{attribute 'strict'}
TYPE E_CSVDataExchangerInsertIntoTableState :
(
	CSV_DATA_EXCHANGER_INSERT_INTO_TABLE_OPEN_FILE 							:= 0,
	CSV_DATA_EXCHANGER_INSERT_INTO_TABLE_WAIT_FOR_OPENING					:= 10,	
	CSV_DATA_EXCHANGER_INSERT_INTO_TABLE_CONV_ONE_RECORD_TO_CSV 			:= 20,	
	CSV_DATA_EXCHANGER_INSERT_INTO_TABLE_WRITE_SINGLE_LINE					:= 30,	
	CSV_DATA_EXCHANGER_INSERT_INTO_TABLE_WAIT_FOR_WRITTING_SINGLE_LINE		:= 40,	
	CSV_DATA_EXCHANGER_INSERT_INTO_TABLE_CLOSE_FILE							:= 50,	
	CSV_DATA_EXCHANGER_INSERT_INTO_TABLE_WAIT_FOR_CLOSING					:= 60,
	CSV_DATA_EXCHANGER_INSERT_INTO_TABLE_WRITTING_DONE						:= 70
);
END_TYPE

(* stored: Version 1.1.0.1, ProductVersion 3.1.4024.12
   DUT E_CSVDataExchangerInsertIntoTableState: Id {0f124281-a07c-42a8-be0f-5cffe8e968d8} *)
